PROGRAM SevenDayCtrl
VAR

	SevenDayOn: fbSevenDaySys;
	SevenDayOff: fbSevenDaySys;

END_VAR

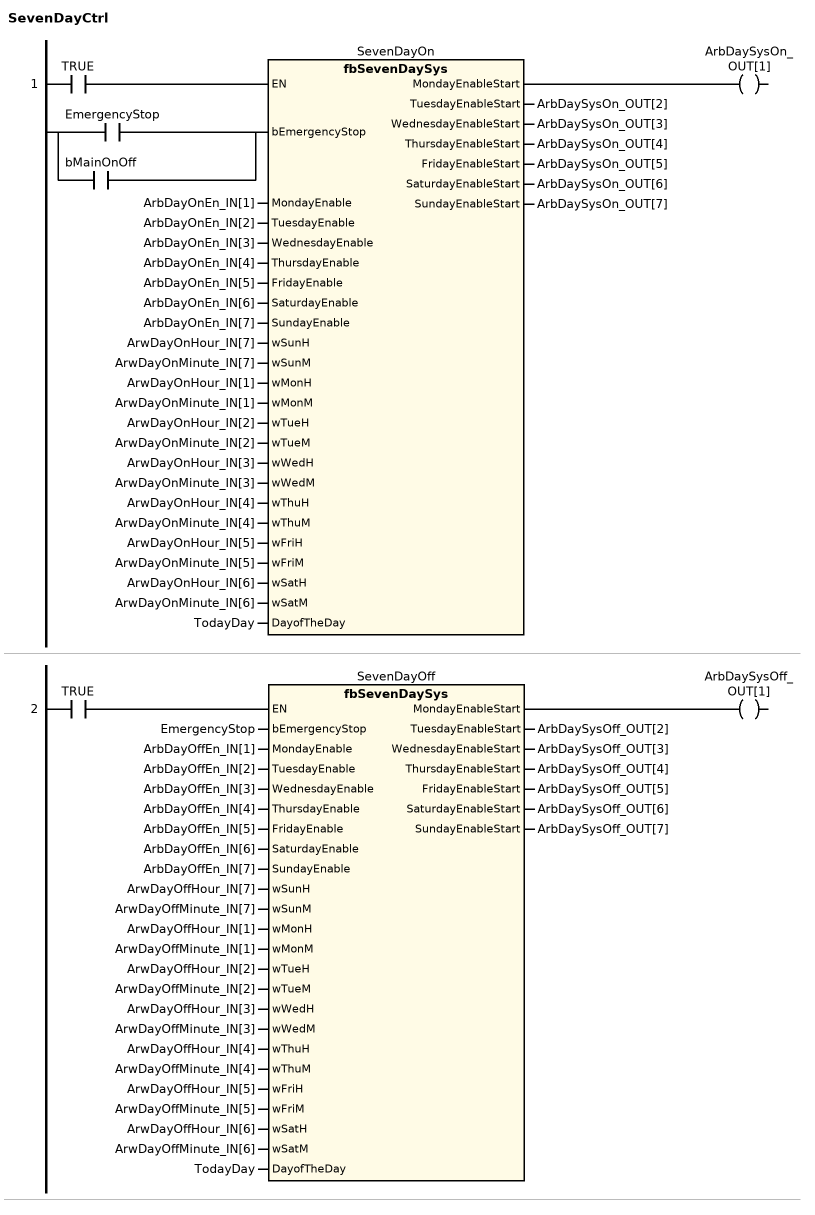
// NETWORK 1
SevenDayOn(
    bEmergencyStop := EmergencyStop OR bMainOnOff,
    MondayEnable := ArbDayOnEn_IN[1],
    TuesdayEnable := ArbDayOnEn_IN[2],
    WednesdayEnable := ArbDayOnEn_IN[3],
    ThursdayEnable := ArbDayOnEn_IN[4],
    FridayEnable := ArbDayOnEn_IN[5],
    SaturdayEnable := ArbDayOnEn_IN[6],
    SundayEnable := ArbDayOnEn_IN[7],
    wSunH := ArwDayOnHour_IN[7],
    wSunM := ArwDayOnMinute_IN[7],
    wMonH := ArwDayOnHour_IN[1],
    wMonM := ArwDayOnMinute_IN[1],
    wTueH := ArwDayOnHour_IN[2],
    wTueM := ArwDayOnMinute_IN[2],
    wWedH := ArwDayOnHour_IN[3],
    wWedM := ArwDayOnMinute_IN[3],
    wThuH := ArwDayOnHour_IN[4],
    wThuM := ArwDayOnMinute_IN[4],
    wFriH := ArwDayOnHour_IN[5],
    wFriM := ArwDayOnMinute_IN[5],
    wSatH := ArwDayOnHour_IN[6],
    wSatM := ArwDayOnMinute_IN[6],
    DayofTheDay := TodayDay,
    TuesdayEnableStart => ArbDaySysOn_OUT[2],
    WednesdayEnableStart => ArbDaySysOn_OUT[3],
    ThursdayEnableStart => ArbDaySysOn_OUT[4],
    FridayEnableStart => ArbDaySysOn_OUT[5],
    SaturdayEnableStart => ArbDaySysOn_OUT[6],
    SundayEnableStart => ArbDaySysOn_OUT[7]); // fbSevenDaySys
ArbDaySysOn_OUT[1] := SevenDayOn.MondayEnableStart;

// NETWORK 2
SevenDayOff(
    bEmergencyStop := EmergencyStop,
    MondayEnable := ArbDayOffEn_IN[1],
    TuesdayEnable := ArbDayOffEn_IN[2],
    WednesdayEnable := ArbDayOffEn_IN[3],
    ThursdayEnable := ArbDayOffEn_IN[4],
    FridayEnable := ArbDayOffEn_IN[5],
    SaturdayEnable := ArbDayOffEn_IN[6],
    SundayEnable := ArbDayOffEn_IN[7],
    wSunH := ArwDayOffHour_IN[7],
    wSunM := ArwDayOffMinute_IN[7],
    wMonH := ArwDayOffHour_IN[1],
    wMonM := ArwDayOffMinute_IN[1],
    wTueH := ArwDayOffHour_IN[2],
    wTueM := ArwDayOffMinute_IN[2],
    wWedH := ArwDayOffHour_IN[3],
    wWedM := ArwDayOffMinute_IN[3],
    wThuH := ArwDayOffHour_IN[4],
    wThuM := ArwDayOffMinute_IN[4],
    wFriH := ArwDayOffHour_IN[5],
    wFriM := ArwDayOffMinute_IN[5],
    wSatH := ArwDayOffHour_IN[6],
    wSatM := ArwDayOffMinute_IN[6],
    DayofTheDay := TodayDay,
    TuesdayEnableStart => ArbDaySysOff_OUT[2],
    WednesdayEnableStart => ArbDaySysOff_OUT[3],
    ThursdayEnableStart => ArbDaySysOff_OUT[4],
    FridayEnableStart => ArbDaySysOff_OUT[5],
    SaturdayEnableStart => ArbDaySysOff_OUT[6],
    SundayEnableStart => ArbDaySysOff_OUT[7]); // fbSevenDaySys
ArbDaySysOff_OUT[1] := SevenDayOff.MondayEnableStart;

END_PROGRAM

(* stored: Version 1.1.0.1, ProductVersion 3.1.4024.12
   POU SevenDayCtrl: Id {0e8ff89c-d1ea-44aa-8c80-961750667d3d}, SpecialFunc None *)
